PROGRAM IrDistanceSensors
VAR
	distanceRaw AT %I* : ARRAY [1..9] OF INT;
	
	distance_mm AT %Q* : ARRAY [1..9] OF REAL;

	i : INT;
END_VAR

FOR  i := 1 TO 9 DO
	distance_mm[i] := IrDistanceFromRaw(distanceRaw[i]);
END_FOR

END_PROGRAM

(* stored: Version 1.1.0.1, ProductVersion 3.1.4024.6
   POU IrDistanceSensors: Id {a7ebd4d1-b79f-44fb-9aa2-85a679c908b8}, SpecialFunc None *)
